FUNCTION_BLOCK Seq_Teile_Hohlen EXTENDS FB_Basis IMPLEMENTS I_Sequenz
VAR_INPUT
	// Prozessparameter		
	Param_StartPos				:sRoboterProzessVariablen;
	Param_Backenbreite			:USINT;
	
	// Objekt-Schnittstellen
	I_Roboter					:I_Objekt_Roboter;
	I_Greifer					:I_Objekt_SmartGreifer;	
	
END_VAR
VAR_OUTPUT
	
END_VAR
VAR
	// Skill-Instanziierung
	Skill_R_P2P				:Skill_Position_anfahren;
	Skill_G_P2P				:Skill_Greifer_Pos_Anfahren;
	
	// Interne Prozessvariablen
	LRobotVar				:sRoboterProzessVariablen;
	LGreiferVar				:sSmartGreiferProzessVariablen;
	LOffsetVar				:LREAL;
	
END_VAR

// Ablauf
ACT_Ablauf();

// Zustandshandling
CASE iState OF
	0:	// BEREIT
		IF bStart THEN
			iState := 1;
		END_IF
	1:	// LAUFEND
		IF eSysCommand = 4 THEN
			bReset := TRUE;
			SFCReset := TRUE;
		END_IF
		
		IF bBeendet OR bReset THEN
			bReset := FALSE;
			SFCReset := FALSE;
			iState := 0;
		END_IF
	2: // ABGESCHLOSSEN
		IF SFCCurrentStep = 'Init' THEN
			iState := 0;
		END_IF
END_CASE

ACTION ACT_Ablauf:
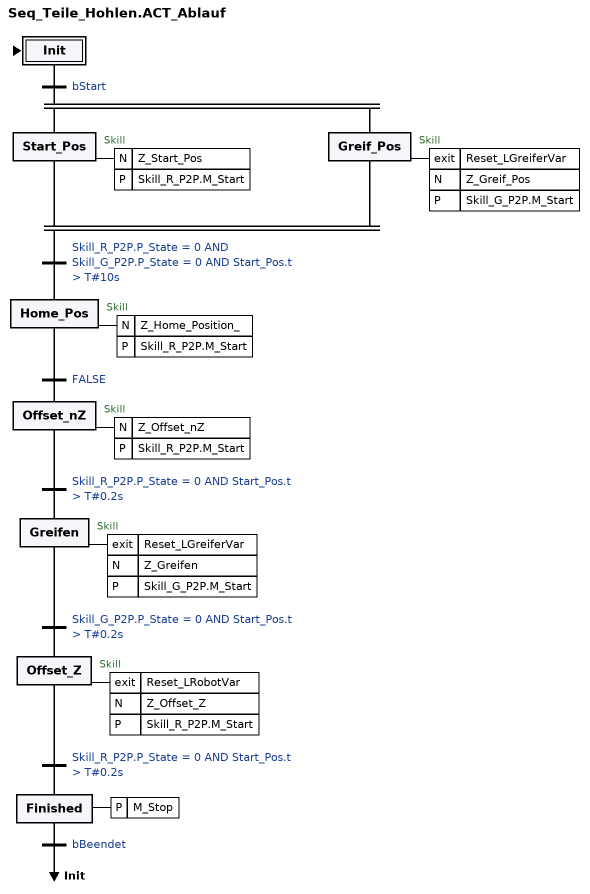
INITIAL_STEP Init:
END_STEP
TRANSITION FROM Init TO (Start_Pos, Greif_Pos)
    := bStart;
END_TRANSITION
// Skill
STEP Start_Pos:
    Z_Start_Pos(N);
    Skill_R_P2P.M_Start(P);
END_STEP
// Skill
STEP Greif_Pos:
    Reset_LGreiferVar(P0);  // exit action
    Z_Greif_Pos(N);
    Skill_G_P2P.M_Start(P);
END_STEP
TRANSITION FROM (Start_Pos, Greif_Pos) TO Home_Pos
    := Skill_R_P2P.P_State = 0 AND Skill_G_P2P.P_State = 0 AND Start_Pos.t > T#10s;
END_TRANSITION
// Skill
STEP Home_Pos:
    Z_Home_Position_(N);
    Skill_R_P2P.M_Start(P);
END_STEP
TRANSITION FROM Home_Pos TO Offset_nZ
    := FALSE;
END_TRANSITION
// Skill
STEP Offset_nZ:
    Z_Offset_nZ(N);
    Skill_R_P2P.M_Start(P);
END_STEP
TRANSITION FROM Offset_nZ TO Greifen
    := Skill_R_P2P.P_State = 0 AND Start_Pos.t > T#0.2s;
END_TRANSITION
// Skill
STEP Greifen:
    Reset_LGreiferVar(P0);  // exit action
    Z_Greifen(N);
    Skill_G_P2P.M_Start(P);
END_STEP
TRANSITION FROM Greifen TO Offset_Z
    := Skill_G_P2P.P_State = 0 AND Start_Pos.t > T#0.2s;
END_TRANSITION
// Skill
STEP Offset_Z:
    Reset_LRobotVar(P0);  // exit action
    Z_Offset_Z(N);
    Skill_R_P2P.M_Start(P);
END_STEP
TRANSITION FROM Offset_Z TO Finished
    := Skill_R_P2P.P_State = 0 AND Start_Pos.t > T#0.2s;
END_TRANSITION
STEP Finished:
    M_Stop(P);
END_STEP
TRANSITION FROM Finished TO Init
    := bBeendet;
END_TRANSITION
// branch label Branch0_ACT_Ablauf
END_ACTION

ACTION Reset_LGreiferVar:
LGreiferVar.F := 0;
LGreiferVar.Geschw := 0;
LGreiferVar.Pos := 0;
END_ACTION

ACTION Reset_LRobotVar:
LRobotVar.q1 := 0;
LRobotVar.q2 := 0;
LRobotVar.q3 := 0;
LRobotVar.q4 := 0;
LRobotVar.q5 := 0;
LRobotVar.q6 := 0;
LRobotVar.v := 0;
LRobotVar.a := 0;
LRobotVar.MoveTyp := 0;
LRobotVar.PosTyp := 0;
END_ACTION

ACTION Z_Greif_Pos:
// Skillaufruf
Skill_G_P2P(eSysCommand := GVL.SystemCommand,
			eSysState := GVL.SystemState,
			Objekt := I_Greifer,
			iErrorID => GVL.ErrorID);
			
// Parameterbestimmung
LGreiferVar.F := 100;
LGreiferVar.Geschw := 100;
LGreiferVar.Pos := Param_Backenbreite;		

// Parameterzuweisung
Skill_G_P2P.P_SGripperParam := LGreiferVar;
END_ACTION

ACTION Z_Greifen:
// Skillaufruf
Skill_G_P2P(eSysCommand := GVL.SystemCommand,
			eSysState := GVL.SystemState,
			Objekt := I_Greifer,
			iErrorID => GVL.ErrorID);
			
// Parameterbestimmung
LGreiferVar.F := 50;
LGreiferVar.Geschw := 50;
LGreiferVar.Pos := 10;		

// Parameterzuweisung
Skill_G_P2P.P_SGripperParam := LGreiferVar;
END_ACTION

ACTION Z_Home_Position_:
// Skillaufruf
Skill_R_P2P(eSysCommand := GVL.SystemCommand,
			eSysState := GVL.SystemState,
			Objekt := I_Roboter,
			iErrorID => GVL.ErrorID);


// Parameterbestimmung			
LRobotVar := PunkteZuweisung_Temp.PHome;
		
// Parameterzuweisung	
Skill_R_P2P.P_RobotParam := LRobotVar;
END_ACTION

ACTION Z_Offset_nZ:
// Skillaufruf
Skill_R_P2P(eSysCommand := GVL.SystemCommand,
			eSysState := GVL.SystemState,
			Objekt := I_Roboter,
			iErrorID => GVL.ErrorID);

// Parameterbestimmung			
LRobotVar.q1 := 0;
LRobotVar.q2 := 0;
LRobotVar.q3 := -0.03;
LRobotVar.q4 := 0;
LRobotVar.q5 := 0;
LRobotVar.q6 := 0;
LRobotVar.v := 0.1;
LRobotVar.a := 0.1;
LRobotVar.MoveTyp := 0;
LRobotVar.PosTyp := 1;

// Parameterzuweisung	
Skill_R_P2P.P_RobotParam := LRobotVar;
END_ACTION

ACTION Z_Offset_Z:
// Skillaufruf
Skill_R_P2P(eSysCommand := GVL.SystemCommand,
			eSysState := GVL.SystemState,
			Objekt := I_Roboter,
			iErrorID => GVL.ErrorID);

// Parameterbestimmung			
LRobotVar.q1 := 0;
LRobotVar.q2 := 0;
LRobotVar.q3 := 0.03;
LRobotVar.q4 := 0;
LRobotVar.q5 := 0;
LRobotVar.q6 := 0;
LRobotVar.v := 0.1;
LRobotVar.a := 0.1;
LRobotVar.MoveTyp := 0;
LRobotVar.PosTyp := 1;
		
// Parameterzuweisung	
Skill_R_P2P.P_RobotParam := LRobotVar;
END_ACTION

ACTION Z_Start_Pos:
// Skillaufruf
Skill_R_P2P(eSysCommand := GVL.SystemCommand,
			eSysState := GVL.SystemState,
			Objekt := I_Roboter,
			iErrorID => GVL.ErrorID);

// Parameterbestimmung			
LRobotVar := Param_StartPos;
		
// Parameterzuweisung	
Skill_R_P2P.P_RobotParam := LRobotVar;
END_ACTION

END_FUNCTION_BLOCK

(* stored: Version 1.1.0.1
   POU Seq_Teile_Hohlen: Id {3ab1661f-bca8-48a2-ae3c-ae654f4f2e0c}, SpecialFunc None
   Folder 00_Resetten: Id {423a6df8-95e5-4bf4-9beb-6956cb2ad30b}
   Folder 01_Zuweisung: Id {1ec76369-d69f-4367-a471-342380850034}
   Action ACT_Ablauf: Id {f6f92059-91e4-4a97-9405-188641de22cc}
   Action Reset_LGreiferVar: Id {9d3ba51b-68db-4969-b0ec-bd6026784695}
   Action Reset_LRobotVar: Id {c7d610f8-338a-4f70-9eb5-d7188d3de136}
   Action Z_Greif_Pos: Id {d3fef3d4-c96d-45ae-8528-42d88906181b}
   Action Z_Greifen: Id {f39cddff-5c7f-43c2-a680-68cd117303fb}
   Action Z_Home_Position_: Id {1c550bea-b9ce-4791-b09b-797d27b9f5fa}
   Action Z_Offset_nZ: Id {e1dacfae-3213-452a-9198-1f4a435392ac}
   Action Z_Offset_Z: Id {1879a83e-38ba-480f-9ce5-5bc8580a54f5}
   Action Z_Start_Pos: Id {60a67d5d-5211-40e2-bdcc-18dbb6c3cfcb} *)
